Fanuc KAREL source: kt00154.KL

-- PROVISIONAL review KL for V770-1; original PC SHA256 27a495942fafd1fa8fcee7350fbb22f13d360951e616628b871d54828a3d2d68
-- Incomplete behavior may be omitted. Consult companion uncertainty JSON. Do not deploy.
PROGRAM KT00154
%NOLOCKGROUP
VAR
  I2 : INTEGER
  OUT : REAL
-- UNRESOLVED_DECL H1 type=002017
BEGIN
  -- UNRESOLVED_PC offsets 5-19; opcodes 2E,22,9D,33,B4
  -- UNRESOLVED_PC offsets 24-35; opcodes 2E,23
  -- UNRESOLVED_PC offsets 40-63; opcodes 22,9D,33,B3,21,55,64,23
  -- UNRESOLVED_PC offsets 68-72; opcodes 7F
END KT00154
